KUKA KRL program: dockon_3.src, dockon_3.dat

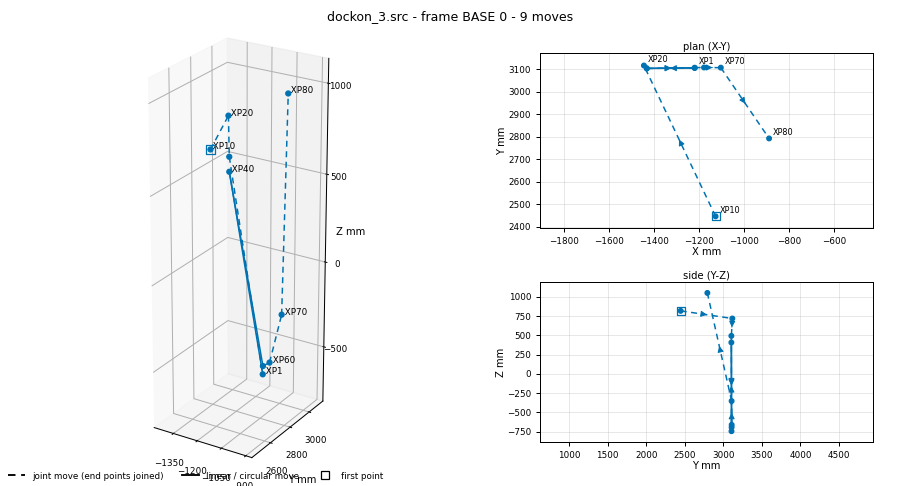
[picture p0: tool path of dockon_3.src in frame BASE 0, 9 of 9 moves have a stored position in this frame; points joined in program order, loops and branches not executed]
--- dockon_3.src ---
&ACCESS RV1
&REL 138
&COMMENT PICKUP GUN 3
DEF DOCKON_3( )
;================================================
; MODEL    :
; IE GROUP :
; STATION  :
; ROBOT    :
; FUNCTION : DOCK ON GUN 3
;================================================
;FOLD INI
;FOLD BASISTECH INI
GLOBAL INTERRUPT DECL 3 WHEN $STOPMESS==TRUE DO IR_STOPM ( )
INTERRUPT ON 3
BAS (#INITMOV,0 )
;ENDFOLD (BASISTECH INI)
;FOLD USER INI
;Make your modifications here
;ENDFOLD (USER INI)
;ENDFOLD (INI)

;FOLD PTP p10  Vel= 100 % H Tool[10]:DOCKING PLATE Base[0];%{PE}%R 5.2.271,%MKUKATPBASIS,%CMOVE,%VPTP,%P 1:PTP, 2:p10, 3:, 5:100, 7:H
$BWDSTART = FALSE
PDAT_ACT=PH
FDAT_ACT=FP10
BAS(#PTP_PARAMS,100)
PTP XP10
;ENDFOLD

;Open flap 3
;FOLD DOCKING.FLAP_OPN 3 ;%{PE}%MKUKATPUSER
DOCKING (#FLAP_OPN ,3)
;ENDFOLD

;FOLD ; Check docking station 3 ready to dock on;%{PE}%R 2.4.14,%MKUKATPBASIS,%CCOMMENT,%VNORMAL,%P 2:Check docking station 3 ready to dock on
;ENDFOLD
DOCKING (#REQ_DOCK_ON ,3)

;FOLD PTP p20 CONT Vel= 100 % H Tool[10]:Docking plaat Base[0];%{PE}%R 5.2.271,%MKUKATPBASIS,%CMOVE,%VPTP,%P 1:PTP, 2:p20, 3:C_PTP, 5:100, 7:H
$BWDSTART = FALSE
PDAT_ACT=PH
FDAT_ACT=FP20
BAS(#PTP_PARAMS,100)
PTP XP20 C_PTP
;ENDFOLD

;FOLD ; Above dock position station 3;%{PE}%R 2.4.14,%MKUKATPBASIS,%CCOMMENT,%VNORMAL,%P 2:Above dock position station 3
;ENDFOLD
;FOLD PTP p30  Vel= 100 % H Tool[10]:Docking plaat Base[0];%{PE}%R 5.2.271,%MKUKATPBASIS,%CMOVE,%VPTP,%P 1:PTP, 2:p30, 3:, 5:100, 7:H
$BWDSTART = FALSE
PDAT_ACT=PH
FDAT_ACT=FP30
BAS(#PTP_PARAMS,100)
PTP XP30
;ENDFOLD


;FOLD PTP P1  Vel= 100 % PDAT1 Tool[3]:Gun 3 Base[0];%{PE}%R 5.4.35,%MKUKATPBASIS,%CMOVE,%VPTP,%P 1:PTP, 2:P1, 3:, 5:100, 7:PDAT1
$BWDSTART=FALSE
PDAT_ACT=PPDAT1
FDAT_ACT=FP1
BAS(#PTP_PARAMS,100)
PTP XP1
;ENDFOLD

;FOLD ; In Dock position Station 3;%{PE}%R 2.4.14,%MKUKATPBASIS,%CCOMMENT,%VNORMAL,%P 2:In Dock position Station 3
;ENDFOLD
;FOLD LIN p40  Vel= 0.2 m/s H Tool[10]:Docking plaat Base[0];%{PE}%R 5.2.271,%MKUKATPBASIS,%CMOVE,%VLIN,%P 1:LIN, 2:p40, 3:, 5:0.2, 7:H
$BWDSTART = FALSE
LDAT_ACT=LH
FDAT_ACT=FP40
BAS(#CP_PARAMS,0.2)
LIN XP40
;ENDFOLD

;FOLD ; Lock Docking plate;%{PE}%R 2.4.14,%MKUKATPBASIS,%CCOMMENT,%VNORMAL,%P 2:Lock Docking plate
;ENDFOLD
DOCKING (#TOOL_LOCK,3)

;FOLD ; Out Docking station 3;%{PE}%R 2.4.14,%MKUKATPBASIS,%CCOMMENT,%VNORMAL,%P 2:Out Docking station 3
;ENDFOLD
;FOLD LIN p50  Vel= 0.2 m/s H Tool[3]:Gun 3 Base[0];%{PE}%R 5.4.35,%MKUKATPBASIS,%CMOVE,%VLIN,%P 1:LIN, 2:p50, 3:, 5:0.2, 7:H
$BWDSTART=FALSE
LDAT_ACT=LH
FDAT_ACT=FP50
BAS(#CP_PARAMS,0.2)
LIN XP50
;ENDFOLD

;FOLD ; Check docking plate close and station 3 ok;%{PE}%R 5.4.35,%MKUKATPBASIS,%CCOMMENT,%VNORMAL,%P 2:Check docking plate close and station 3 ok
;ENDFOLD
DOCKING (#CHK_TOOL_ON,3)

;FOLD PTP p60 CONT Vel= 100 % H Tool[3]:Gun 3 Base[0];%{PE}%R 5.4.35,%MKUKATPBASIS,%CMOVE,%VPTP,%P 1:PTP, 2:p60, 3:C_PTP, 5:100, 7:H
$BWDSTART=FALSE
PDAT_ACT=PH
FDAT_ACT=FP60
BAS(#PTP_PARAMS,100)
PTP XP60 C_PTP
;ENDFOLD
;FOLD PTP p70 CONT Vel= 100 % H Tool[3]:Gun 3 Base[0];%{PE}%R 5.4.35,%MKUKATPBASIS,%CMOVE,%VPTP,%P 1:PTP, 2:p70, 3:C_PTP, 5:100, 7:H
$BWDSTART=FALSE
PDAT_ACT=PH
FDAT_ACT=FP70
BAS(#PTP_PARAMS,100)
PTP XP70 C_PTP
;ENDFOLD
;FOLD PTP p80  Vel= 100 % H Tool[3]:Gun 3 Base[0];%{PE}%R 5.4.35,%MKUKATPBASIS,%CMOVE,%VPTP,%P 1:PTP, 2:p80, 3:, 5:100, 7:H
$BWDSTART=FALSE
PDAT_ACT=PH
FDAT_ACT=FP80
BAS(#PTP_PARAMS,100)
PTP XP80
;ENDFOLD

END

--- dockon_3.dat ---
&ACCESS RV1
&REL 138
&COMMENT PICKUP GUN 3
DEFDAT  DOCKON_3
;FOLD EXTERNAL DECLARATIONS;%{PE}%MKUKATPBASIS,%CEXT,%VCOMMON,%P
;FOLD GRIPPERTECH EXT
EXT  H50 (INT  :IN,INT  :IN,INT  :IN,GRP_TYP  :IN )
;ENDFOLD (GRIPPERTECH EXT)
;FOLD SPOTTECH EXT
EXT  USERSPOT (S_COMMAND  :IN,SPOT_TYPE  :IN )
;ENDFOLD (SPOTTECH EXT)
;FOLD BASISTECH EXT;%{PE}%MKUKATPBASIS,%CEXT,%VEXT,%P
EXT  BAS (BAS_COMMAND  :IN,REAL  :IN )
DECL INT SUCCESS
;ENDFOLD (BASISTECH EXT)
;FOLD USER EXT;%{E}%MKUKATPUSER,%CEXT,%VEXT,%P
;Make here your modifications
;ENDFOLD (USER EXT)
;ENDFOLD (EXTERNAL DECLERATIONS)
DECL GRP_TYP GCONT={G_APO #YES,TIME 0.0,CTRL #OFF,DLY 0,DST 0}
DECL GRP_TYP GGDAT={G_APO #NO,TIME 0.0,CTRL #OFF,DLY 0,DST 1}
;*      FDAT Declarations     *

;******************************
;*     E6POS Declarations     *
;******************************

DECL E6POS XP10={X -1127.36902,Y 2445.76807,Z 816.869385,A -45.7330017,B 0.4947837,C 179.7724,S 2,T 11,E1 -1181.96399,E2 0.0,E3 0.0,E4 0.0,E5 0.0,E6 0.0}
DECL E6POS XP20={X -1446.12402,Y 3116.53906,Z 717.922974,A 58.8610001,B -0.318507999,C -179.604202,S 2,T 3,E1 -1703.68103,E2 0.0,E3 0.0,E4 0.0,E5 0.0,E6 0.0}
DECL E6POS XP30={X -1433.29297,Y 3103.76904,Z 492.324188,A 58.8653107,B -0.296647787,C -179.599304,S 2,T 3,E1 -1703.68103,E2 0.0,E3 0.0,E4 0.0,E5 0.0,E6 0.0}
DECL E6POS XP40={X -1433.297,Y 3103.77197,Z 406.572693,A 58.865181,B -0.296665102,C -179.598999,S 2,T 3,E1 -1703.68103,E2 0.0,E3 0.0,E4 0.0,E5 0.0,E6 0.0}
DECL E6POS XP50={X -1220.43506,Y 3106.93091,Z -694.426208,A -13.5916004,B 72.6322479,C -12.8654499,S 2,T 3,E1 -1703.68298,E2 0.0,E3 0.0,E4 0.0,E5 0.0,E6 0.0}
DECL E6POS XP60={X -1178.72095,Y 3107.79907,Z -662.205017,A -13.5877895,B 72.6321716,C -12.8613501,S 2,T 3,E1 -1703.68298,E2 0.0,E3 0.0,E4 0.0,E5 0.0,E6 0.0}
DECL E6POS XP70={X -1104.13306,Y 3107.021,Z -353.061005,A -13.5874701,B 72.6343613,C -12.8619604,S 2,T 3,E1 -1703.68506,E2 0.0,E3 0.0,E4 0.0,E5 0.0,E6 0.0}
DECL E6POS XP80={X -889.438477,Y 2792.34302,Z 1049.42505,A -106.691704,B 85.8009872,C -106.606796,S 2,T 11,E1 -1703.68701,E2 0.0,E3 0.0,E4 0.0,E5 0.0,E6 0.0}

;******************************
;*     FDAT Declarations      *
;******************************

DECL FDAT FP10={TOOL_NO 10,BASE_NO 0,IPO_FRAME #BASE}
DECL FDAT FP20={TOOL_NO 10,BASE_NO 0,IPO_FRAME #BASE}
DECL FDAT FP30={TOOL_NO 10,BASE_NO 0,IPO_FRAME #BASE}
DECL FDAT FP40={TOOL_NO 10,BASE_NO 0,IPO_FRAME #BASE}
DECL FDAT FP50={TOOL_NO 3,BASE_NO 0,IPO_FRAME #BASE}
DECL FDAT FP60={TOOL_NO 3,BASE_NO 0,IPO_FRAME #BASE}
DECL FDAT FP70={TOOL_NO 3,BASE_NO 0,IPO_FRAME #BASE}
DECL FDAT FP80={TOOL_NO 3,BASE_NO 0,IPO_FRAME #BASE}

;******************************
;*  PDAT & LDAT Declarations  *
;******************************

DECL PDAT PH={VEL 100.0,ACC 100.0,APO_DIST 100.0}
DECL LDAT LH={VEL 2.0,ACC 100.0,APO_DIST 100.0,APO_FAC 50.0,ORI_TYP #VAR}

DECL E6POS XP1={X -1220.39795,Y 3105.43091,Z -744.515076,A -13.7468996,B 72.6471634,C -12.8395901,S 2,T 3,E1 -1701.58704,E2 0.0,E3 0.0,E4 0.0,E5 0.0,E6 0.0}
DECL FDAT FP1={TOOL_NO 3,BASE_NO 0,IPO_FRAME #BASE,POINT2[] " "}
DECL PDAT PPDAT1={VEL 100.0,ACC 100.0,APO_DIST 100.0}
ENDDAT
